// SIMATIC STEP 7 (V5.x) project TEMA 8 EJERCICIO 3
// CPU: CPU313 C-2 DP(1)
// station: P_ADR_BUS
// station: Hardware
// station: Equipo SIMATIC 300
// program: Programa S7(1)

SYMBOL_TABLE
""		
""		
"FLANCO"	DB 1	DB 1
"MANIOBRA"	DB 2	DB 2
"P PARO"	I 0.0	BOOL
"P MARCHA"	I 0.1	BOOL
"RELE TERMICO"	I 0.2	BOOL
"Cycle Execution"	OB 1	OB 1
"LED PARO"	Q 0.0	BOOL
"V L U1-V1-W1"	Q 0.1	BOOL
"V R U2-V2-W2"	Q 0.2	BOOL
"V R CORTOCIRQUITADO"	Q 0.3	BOOL
"LED MARCHA"	Q 0.4	BOOL
"LED AVERIA"	Q 0.5	BOOL
"VAT_1"	VAT 1	
END_SYMBOL_TABLE

DATA_BLOCK "FLANCO"	// DB 1
VERSION : 0.1
  STRUCT
   MARCA0 : BOOL ;
   MARCA1 : BOOL ;
   MARCA2 : BOOL ;
   MARCA3 : BOOL ;
   MARCA4 : BOOL ;
   MARCA5 : BOOL ;
   MARCA6 : BOOL ;
   MARCA7 : BOOL ;
   MARCA10 : BOOL ;
   MARCA11 : BOOL ;
   MARCA12 : BOOL ;
   MARCA13 : BOOL ;
   MARCA14 : BOOL ;
   MARCA15 : BOOL ;
   MARCA16 : BOOL ;
   MARCA17 : BOOL ;
  END_STRUCT ;	
BEGIN
END_DATA_BLOCK

DATA_BLOCK "MANIOBRA"	// DB 2
VERSION : 0.1
  STRUCT
   MARCA0 : BOOL ;
   MARCA1 : BOOL ;
   MARCA2 : BOOL ;
   MARCA3 : BOOL ;
   MARCA4 : BOOL ;
   MARCA5 : BOOL ;
   MARCA6 : BOOL ;
   MARCA7 : BOOL ;
  END_STRUCT ;	
BEGIN
END_DATA_BLOCK

ORGANIZATION_BLOCK "Cycle Execution"	// OB 1
TITLE = "Main Program Sweep (Cycle)"
//ARRANQUE DHALANDER CON ACTIVACION TEMPORIZADA PARA CAMBIO DE VELOCIDAD
VERSION : 0.1
VAR_TEMP
  OB1_EV_CLASS : BYTE ;	//Bits 0-3 = 1 (Coming event), Bits 4-7 = 1 (Event class 1)
  OB1_SCAN_1 : BYTE ;	//1 (Cold restart scan 1 of OB 1), 3 (Scan 2-n of OB 1)
  OB1_PRIORITY : BYTE ;	//Priority of OB Execution
  OB1_OB_NUMBR : BYTE ;	//1 (Organization block 1, OB1)
  OB1_RESERVED_1 : BYTE ;	//Reserved for system
  OB1_RESERVED_2 : BYTE ;	//Reserved for system
  OB1_PREV_CYCLE : INT ;	//Cycle time of previous OB1 scan (milliseconds)
  OB1_MIN_CYCLE : INT ;	//Minimum cycle time of OB1 (milliseconds)
  OB1_MAX_CYCLE : INT ;	//Maximum cycle time of OB1 (milliseconds)
  OB1_DATE_TIME : DATE_AND_TIME ;	//Date and time OB1 started
END_VAR
BEGIN
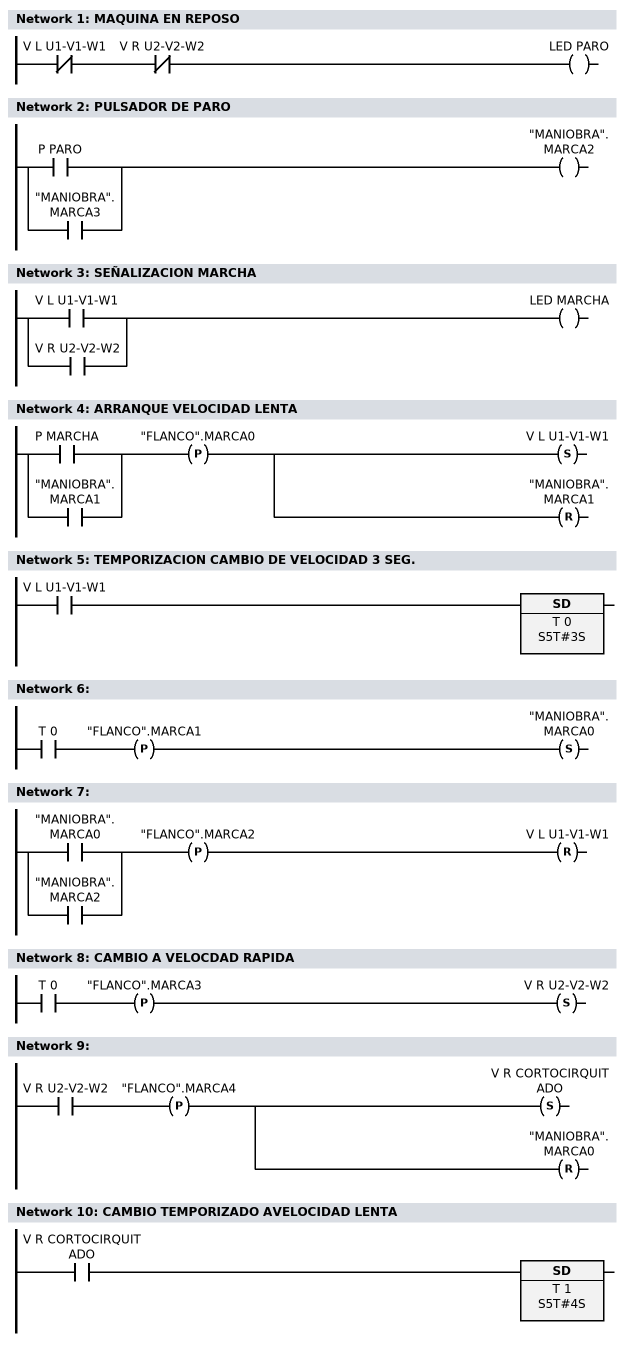
NETWORK
TITLE = MAQUINA EN REPOSO 
//SEÑALIZACION LED DE PARO
      AN    "V L U1-V1-W1";
      AN    "V R U2-V2-W2";
      =     "LED PARO";
NETWORK
TITLE = PULSADOR DE PARO
//POSICION DE REPOSO RESET V LENTA Y V RAPIDA MEDIANTE MARCA MANOBRA 2
      O     "P PARO";
      O     "MANIOBRA".MARCA3;
      =     "MANIOBRA".MARCA2;
NETWORK
TITLE = SEÑALIZACION MARCHA 
//ESTARA ENCENDIDA SIEMPRE QUE HALLA FUNCIONANDO UNA DE LAS DOS VELOCIDADES
      O     "V L U1-V1-W1";
      O     "V R U2-V2-W2";
      =     "LED MARCHA";
NETWORK
TITLE = ARRANQUE VELOCIDAD LENTA
//P MARCHA ALIMENTACION U1-V1-W1 
      A(;
      O     "P MARCHA";
      O     "MANIOBRA".MARCA1;
      );
      FP    "FLANCO".MARCA0;
      S     "V L U1-V1-W1";
      R     "MANIOBRA".MARCA1;
NETWORK
TITLE = TEMPORIZACION CAMBIO DE VELOCIDAD 3 SEG.
//ALIMENTACION TEMPORIZADOR A LA CONEXION T0 (SE)
      A     "V L U1-V1-W1";
      L     S5T#3S;
      SD    T 0;
NETWORK
TITLE =
//CONTACTO TEMPORIZADO ACTIVA MARCA0 DE MANOIOBRA
      A     T 0;
      FP    "FLANCO".MARCA1;
      S     "MANIOBRA".MARCA0;
NETWORK
TITLE =
//MARCA0 MANIOBRA DESACTIVA LENTA 
      A(;
      O     "MANIOBRA".MARCA0;
      O     "MANIOBRA".MARCA2;
      );
      FP    "FLANCO".MARCA2;
      R     "V L U1-V1-W1";
NETWORK
TITLE = CAMBIO A VELOCDAD RAPIDA
//MARCA0 MANIOBRA ACTIVA U2-V2-W2
      A     T 0;
      FP    "FLANCO".MARCA3;
      S     "V R U2-V2-W2";
NETWORK
TITLE =
//ACTO SEGUIDO SE CORTOCIRQUITA LOS BORNES 
      A     "V R U2-V2-W2";
      FP    "FLANCO".MARCA4;
      S     "V R CORTOCIRQUITADO";
      R     "MANIOBRA".MARCA0;
NETWORK
TITLE = CAMBIO TEMPORIZADO AVELOCIDAD LENTA
//ALIMENTACION TEMPORIZADOR 4 SEG.
      A     "V R CORTOCIRQUITADO";
      L     S5T#4S;
      SD    T 1;
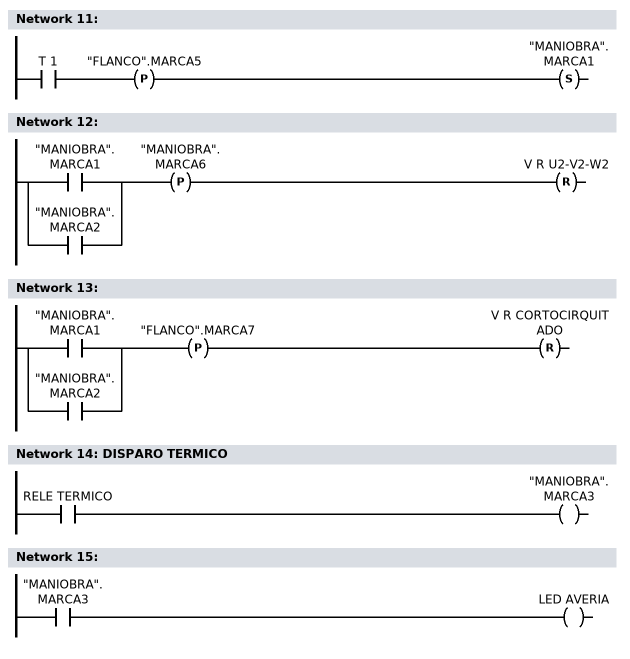
NETWORK
TITLE =
//CONTACTO TEMPORIZADO CONECTA MARCA MANIOBA 1
      A     T 1;
      FP    "FLANCO".MARCA5;
      S     "MANIOBRA".MARCA1;
NETWORK
TITLE =
//MARCA 1 MANIOBRA DESCONECTA U2-V2-W2
      A(;
      O     "MANIOBRA".MARCA1;
      O     "MANIOBRA".MARCA2;
      );
      FP    "MANIOBRA".MARCA6;
      R     "V R U2-V2-W2";
NETWORK
TITLE =
//MARCA 1 MANIOBRA DESCONECTA CORTOCIRQUITADO
      A(;
      O     "MANIOBRA".MARCA1;
      O     "MANIOBRA".MARCA2;
      );
      FP    "FLANCO".MARCA7;
      R     "V R CORTOCIRQUITADO";
NETWORK
TITLE = DISPARO TERMICO 
//LLEVA EL PROGRAMA A SU ESTADO INCIAL Y ENCIENDE LED AVERIA 
      A     "RELE TERMICO";
      =     "MANIOBRA".MARCA3;
NETWORK
TITLE =
      A     "MANIOBRA".MARCA3;
      =     "LED AVERIA";
END_ORGANIZATION_BLOCK
